FUNCTION_BLOCK FlowCalSequence
VAR_INPUT
	start : BOOL := FALSE;  //command to start
	setSpeedDuration : TIME := T#15S;  //Time to allow flow to stabilize before starting run
	runTestDuration : TIME := T#3M; //Time to collect liquid on the scale
	runTestWeight : LREAL := 20.0; // run for 100 grams minimum quantity of fluid on the scale for a completed flowrate
	autoAdvance : BOOL := TRUE; //Determines if the test should automatically start the next flowrate.  Sometimes the flow is too much and the collection vessel has to be emptied
	tubingType :INT := 14;
END_VAR
VAR_IN_OUT
	fq : FQ1; //flow totalizer
	pump : sMasterflexPort;
	FTOLS: OLSResult;
	pumpOLS: OLSResult;
END_VAR
VAR_OUTPUT
	startTimes : ARRAY[1..100] OF ULINT;
	endTimes : ARRAY[1..100] OF ULINT;
	flowTotal : ARRAY[1..100] OF LREAL;
	weight : ARRAY[1..100] OF LREAL;
	flowRate : ARRAY[1..100] OF LREAL;
	scaleRate : ARRAY[1..100] OF LREAL;
	calibrationStatus : UINT := 0;
END_VAR
VAR
	i : UINT := 0; // index
	n : UINT := 24;  //number of points to test
	t : LREAL := 0.0; //temporary variable
	tol : LREAL := 5.0;  //tolerance of the zeroing - weight must be below this to have successfully zero'd
	R2Tol : LREAL := 0.95; //tolerance of the OLS fit
	flowCalMTol : LREAL := 0.05; //tolerance for slope
	flowCalBTol : LREAL := 0.05; //tolerance for intercept
	OLSFlowTemp : OLSResult;
	OLSPumpTemp : OLSResult;
	sp : ARRAY [1..100] OF LREAL := [10.0, 20.0, 30.0, 40.0, 50.0, 60.0, 70.0, 80.0, 90.0, 100.0, 
                                    125.0, 150.0, 175.0, 200.0, 225.0, 250.0, 275.0, 300.0, 350.0, 400.0,
                                    450.0, 500.0, 550.0, 600.0, 0.0, 0.0, 0.0, 0.0, 0.0, 0.0,
                                    0.0, 0.0, 0.0, 0.0, 0.0, 0.0, 0.0, 0.0, 0.0, 0.0,
                                    0.0, 0.0, 0.0, 0.0, 0.0, 0.0, 0.0, 0.0, 0.0, 0.0,
                                    0.0, 0.0, 0.0, 0.0, 0.0, 0.0, 0.0, 0.0, 0.0, 0.0,
                                    0.0, 0.0, 0.0, 0.0, 0.0, 0.0, 0.0, 0.0, 0.0, 0.0,
                                    0.0, 0.0, 0.0, 0.0, 0.0, 0.0, 0.0, 0.0, 0.0, 0.0,
                                    0.0, 0.0, 0.0, 0.0, 0.0, 0.0, 0.0, 0.0, 0.0, 0.0,
                                    0.0, 0.0, 0.0, 0.0, 0.0, 0.0, 0.0, 0.0, 0.0, 0.0
									];

	setSpeed : SFCStepType;
	runTest : SFCStepType;
	recordTest : SFCStepType;
	calcCalibration : SFCStepType;
END_VAR

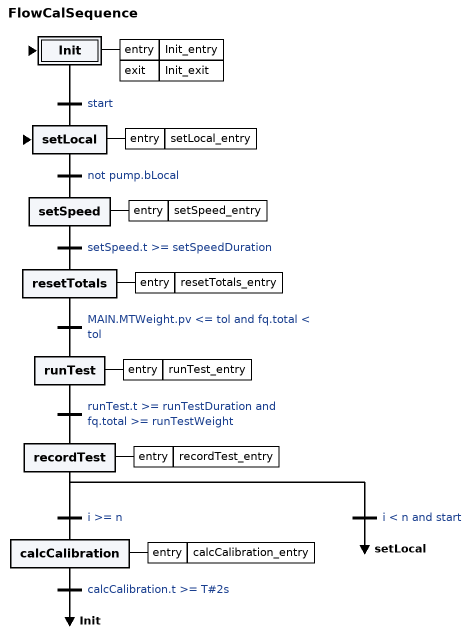
INITIAL_STEP Init:
    Init_entry(P1);  // entry action
    Init_exit(P0);  // exit action
END_STEP
TRANSITION FROM Init TO setLocal
    := start;
END_TRANSITION
STEP setLocal:
    setLocal_entry(P1);  // entry action
END_STEP
TRANSITION FROM setLocal TO setSpeed
    := not pump.bLocal;
END_TRANSITION
STEP setSpeed:
    setSpeed_entry(P1);  // entry action
END_STEP
TRANSITION FROM setSpeed TO resetTotals
    := setSpeed.t >= setSpeedDuration;
END_TRANSITION
STEP resetTotals:
    resetTotals_entry(P1);  // entry action
END_STEP
TRANSITION FROM resetTotals TO runTest
    := MAIN.MTWeight.pv <= tol and fq.total < tol;
END_TRANSITION
STEP runTest:
    runTest_entry(P1);  // entry action
END_STEP
TRANSITION FROM runTest TO recordTest
    := runTest.t >= runTestDuration and fq.total >= runTestWeight;
END_TRANSITION
STEP recordTest:
    recordTest_entry(P1);  // entry action
END_STEP
TRANSITION FROM recordTest TO calcCalibration
    := i >= n;
END_TRANSITION
STEP calcCalibration:
    calcCalibration_entry(P1);  // entry action
END_STEP
TRANSITION FROM recordTest TO setLocal
    := i < n and start;
END_TRANSITION
TRANSITION FROM calcCalibration TO Init
    := calcCalibration.t >= T#2s;
END_TRANSITION

ACTION resetTotals_entry:
fq.resetRQ := TRUE; //reset the totalizer
MAIN.MTSendString := 'ZI$0D$0A';  //Zero Immediately the scale
END_ACTION

ACTION Init_exit:
FOR i := 1 TO n DO
	startTimes[i] := 0;
	endTimes[i] := 0;
	flowTotal[i] := 0.0;
	weight[i] := 0.0;
	flowRate[i] := 0.0;	
	scaleRate[i] := 0.0;	
END_FOR
i := 0;
calibrationStatus := 2; //In process
END_ACTION

ACTION setSpeed_entry:
//Send speed setpoint
IF sp[i] > 0.1 THEN
	pump.nRun_RQ := 1; //start pump
	pump.fSpeedSP_RQ := sp[i];
ELSE
	pump.nRun_RQ := 0; //stop pump
	pump.fSpeedSP_RQ := 0.0;
END_IF
END_ACTION

ACTION runTest_entry:
MAIN.MTSendString := 'SIR$0D$0A'; //Send weight value Immediately and Repeat
startTimes[i] := unixTime;
END_ACTION

ACTION setLocal_entry:
i := i + 1;
IF pump.bLocal THEN
	pump.nLocal_RQ := 0;  //put pump in remote
END_IF
END_ACTION

ACTION Init_entry:
//reset for next calibration
start := FALSE;
END_ACTION

ACTION calcCalibration_entry:
//Stop pump
pump.nRun_RQ := 0; //stop pump

//run data analysis to determine new calibration values
//Check fit of flow data vs. scale data
OLSFlowTemp := ols(x := flowRate, y := scaleRate, length := n);
//Check fit of pump speed data vs. scale data
OLSPumpTemp := ols(x := scaleRate, y := sp, length := n);

//Determine maximum x value of flow data, this is just for the test of intercept
//Expect intercept to be 'near 0.0', so knowing the range of x values is
//necessary to determine what is 'close'
t := 0.0;
FOR i := 1 TO n DO
	t := MAX(t, flowRate[i]);	
END_FOR
IF t = 0.0 THEN //ensure no divide by zero
	t := 1.0;
END_IF

//Check Linearity, slope, and intercept (range and zero)
IF OLSFlowTemp.status <> 0 OR 							//OLS failed
		OLSFlowTemp.R2 < R2Tol OR 						//Not a good line fit
		ABS(1-OLSFlowTemp.m) > flowCalMTol OR  			//Slope not close to 1
		ABS(OLSFlowTemp.b/t) > flowCalBTol THEN			//Intercept is greater than tolerance % of scale
	calibrationStatus := 3; //Failed FT calibration
ELSE
	// Check for pump speed vs. flow 
	IF OLSFlowTemp.status <> 0 OR 						//OLS failed
			OLSFlowTemp.R2 < R2Tol THEN					//Not a good line fit
		calibrationStatus := 4; //Failed pump speed calibration
	ELSE
		calibrationStatus := 1; //Success
		//set both calibrations
		FTOLS := OLSFlowTemp;
		pumpOLS := OLSPumpTemp;  //All checks were good, the calibration is successful.
	END_IF
END_IF
END_ACTION

ACTION recordTest_entry:
endTimes[i] := unixTime;
flowTotal[i] := fq.total;
weight[i] := MAIN.MTWeight.pv;
t := ULINT_TO_LREAL(endTimes[i] - startTimes[i])/1000.0/60.0; //Test duration in minutes
flowRate[i] := flowTotal[i]/t;
scaleRate[i] := weight[i]/t;
IF NOT autoAdvance THEN
	start := FALSE;
END_IF
END_ACTION

END_FUNCTION_BLOCK

(* stored: Version 1.1.0.1, ProductVersion 3.1.0.36
   POU FlowCalSequence: Id {83b04da5-4821-41fa-ac5d-388083e3421e}, SpecialFunc None
   Action resetTotals_entry: Id {04f7def1-f0b6-493d-b18d-42499d2857cc}
   Action Init_exit: Id {32d2533a-d29b-49d4-8e13-63f6c5c2f6e6}
   Action setSpeed_entry: Id {86c1a5e6-debf-4299-97b9-6ab248372f10}
   Action runTest_entry: Id {924250a1-661d-4de0-beaa-23db96c68379}
   Action setLocal_entry: Id {9dbc17ea-44c8-4f1e-bc27-af6a50ca39a1}
   Action Init_entry: Id {ce2cb565-304d-4a9c-ae51-6761afdde65a}
   Action calcCalibration_entry: Id {d1f1becf-b35a-485b-8d31-26a574435737}
   Action recordTest_entry: Id {e6067b70-2130-4502-976d-7f15f6878987} *)
